Fanuc KAREL source: wasymfltrenb.kl

PROGRAM wasymfltrenb
%NOLOCKGROUP
VAR
  p : POSITION
  q : POSITION
  i : INTEGER
  r : REAL
BEGIN
  WITH $ASYMFLTRENB = TRUE MOVE TO p
END wasymfltrenb
